Staubli VAL3: remGetArmStat.pgx

program remGetArmStat(string& sReturn[] (dimensions=1))
begin
  // Get whether power is enabled or disabled
  //
  logMsg("call remGetArmStat")
  if isPowered()
    sReturn="GETARMSTAT ENABLED"
  else
    sReturn="GETARMSTAT DISABLED"
  endIf
end
